// TIA Portal V16 export
// export: Created 2021-11-12T13:32:44.479513Z, ExportSetting WithDefaults, DisplayName Totally Integrated Automation Portal, DisplayVersion V16 Update 3, DisplayName TIA Portal Version Control Interface, DisplayVersion V16 Update 2, DisplayName TIA Portal Openness, DisplayVersion V16 Update 3, DisplayName SINAMICS Startdrive Advanced, DisplayVersion V16 Update 5, DisplayName SINAMICS Startdrive G130, G150, S120, S150, SINAMICS MV, S210, DisplayVersion V16 Update 5, DisplayName SINAMICS Startdrive G110M, G120, G120C, G120D, G120P, G115D, DisplayVersion V16 Update 5, DisplayName STEP 7 Professional, DisplayVersion V16 Update 3, DisplayName STEP 7 Safety, DisplayVersion V16, DisplayName WinCC UA Professional, DisplayVersion V16 Update 3
FUNCTION_BLOCK "StationBSN3"   // FB46, LAD
{ S7_Optimized_Access := 'TRUE' }
VERSION : 0.1
// stored: AutoNumber true, IsIECCheckEnabled false, IsRetainMemResEnabled false, MemoryReserve 100, SetENOAutomatically false, UDAEnableTagReadback false
   VAR_INPUT
      IS_Inputs : "UDT_COMM_BSN3_CRS";   // Inputs from owens PLC
   END_VAR
   VAR_OUTPUT
      OS_Outputs : "UDT_COMM_CRS_BSN3";   // Outputs to owens PLC
      OS_Status : "UDT_BSN3_Status_specific";
   END_VAR
   VAR
      SF_TON_Tact : TON_TIME;
      SF_TON_1 { S7_SetPoint := 'True'} : TON_TIME;
      SF_Alarm1 : "STD_DI_Mon";
      SF_Alarm2 : "STD_DI_Mon";
      SF_Alarm3 : "STD_DI_Mon";
      SF_Alarm4 : "STD_DI_Mon";
      SF_Alarm5 : "STD_DI_Mon";
      SF_Alarm6 : "STD_DI_Mon";
      SF_Alarm7 : "STD_DI_Mon";
      SF_Alarm8 : "STD_DI_Mon";
      SF_CL01_Alarm { S7_SetPoint := 'True'} : "STD_DI_Mon";
      SF_CL01_Warning { S7_SetPoint := 'True'} : "STD_DI_Mon";
      SF_BoxPartCounter { S7_SetPoint := 'True'} : "STD_PartCounter";
      SS_Edge { S7_SetPoint := 'True'} : Array[0..15] of Bool;   // Edge evalution
      SS_ParamTemp : Struct
         PartType : Int;   // Production type
         SPBurnerHigh : Int := 0;   // setpoint burner high [mm]
         SPTempSetpointZ1 : Int := 0;   // temperature setpoint in zone 1 [°C]
         SPTempSetpointZ2 : Int := 0;   // temperature setpoint in zone 2 [°C]
         SPTempSetpointZ3 : Int := 0;   // temperature setpoint in zone 3 [°C]
         SPTempSetpointZ4 : Int := 0;   // temperature setpoint in zone 4 [°C]
         SPTempSetpointZ5 : Int := 0;   // temperature setpoint in zone 5 [°C]
         SPTempSetpointZ6 : Int := 0;   // temperature setpoint in zone 5 [°C]
         SPTempSetpointZ7 : Int := 0;   // temperature setpoint in zone 5 [°C]
         ActPartTime : Int;   // actual setpoint of time in furnace according to belt speed [min]
      END_STRUCT;
      SB1BoxExchangeReq { S7_SetPoint := 'True'} : Bool;
      SB1ReqBlockBeltMtion : Bool;   // Button request to block belt motion
      SB1ReqBlockBeltMtion_Aux : Bool;
      SB1ParamChanged : Bool;   // Production paramaters changed trigger
      ST_RunConv { S7_SetPoint := 'True'} : TOF_TIME;
   END_VAR
   VAR_TEMP
      TS_ParamTemp : Struct
         PartType : Int;   // Production type
         SPBurnerHigh : Int;   // setpoint burner high [mm]
         SPTempSetpointZ1 : Int;   // temperature setpoint in zone 1 [°C]
         SPTempSetpointZ2 : Int;   // temperature setpoint in zone 2 [°C]
         SPTempSetpointZ3 : Int;   // temperature setpoint in zone 3 [°C]
         SPTempSetpointZ4 : Int;   // temperature setpoint in zone 4 [°C]
         SPTempSetpointZ5 : Int;   // temperature setpoint in zone 5 [°C]
         SPTempSetpointZ6 : Int;   // temperature setpoint in zone 5 [°C]
         SPTempSetpointZ7 : Int;   // temperature setpoint in zone 5 [°C]
         ActPartTime : Int;   // actual setpoint of time in furnace according to belt speed [min]
      END_STRUCT;
      TI_NoOfParts : Int;   // Number of parts before press
      TB1BoxFull : Bool;   // Box is full
      TB1PwrOk : Bool;
      TB1BeltMtionBlock : Bool;   // Belt motion blocking
      TB1ReqBlockBeltMtion : Bool;
      TB1ReqOnePart : Bool;   // Request to eject one part
      TB1ReqAllParts : Bool;   // Request to eject all parts in row
      TB1SetParam : Bool;   // Set loaded parameters memory
   END_VAR
   VAR_TEMP   // added for the SCL form of the ladder/FBD networks
      _w1 : Bool;
      _w2 : Bool;
   END_VAR
BEGIN

REGION Network 1: Copy In/Out variables to temporary variables
END_REGION

REGION Network 2: *************** Alarms ***************
END_REGION

REGION Network 3: Power OK
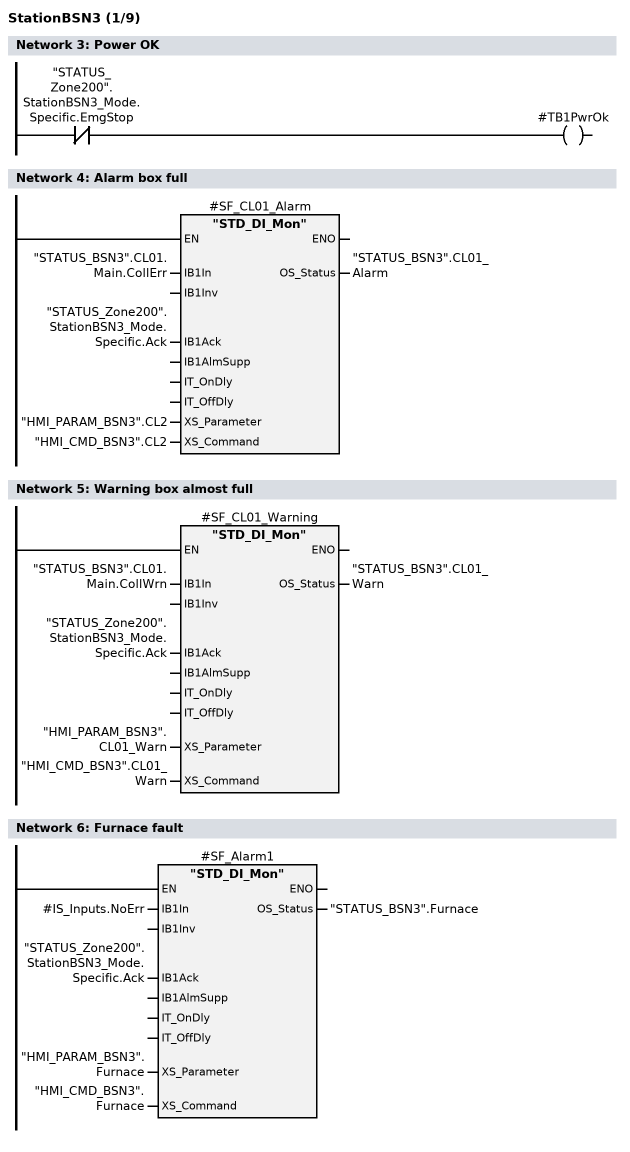
   RUNG wire#powerrail
      I_Contact( "STATUS_Zone200".StationBSN3_Mode.Specific.EmgStop )
      Coil( #TB1PwrOk )
   END_RUNG
   // the same network as SCL:
   #TB1PwrOk := NOT "STATUS_Zone200".StationBSN3_Mode.Specific.EmgStop;
END_REGION

REGION Network 4: Alarm box full
   RUNG wire#powerrail
      #SF_CL01_Alarm(IB1In := "STATUS_BSN3".CL01.Main.CollErr, IB1Inv :=, IB1Ack := "STATUS_Zone200".StationBSN3_Mode.Specific.Ack, IB1AlmSupp :=, IT_OnDly :=, IT_OffDly :=, XS_Parameter := "HMI_PARAM_BSN3".CL2, XS_Command := "HMI_CMD_BSN3".CL2, OS_Status => "STATUS_BSN3".CL01_Alarm)
   END_RUNG
   // the same network as SCL:
   #SF_CL01_Alarm(IB1In := "STATUS_BSN3".CL01.Main.CollErr,   // "STD_DI_Mon"
                  IB1Ack := "STATUS_Zone200".StationBSN3_Mode.Specific.Ack,
                  XS_Parameter := "HMI_PARAM_BSN3".CL2,
                  XS_Command := "HMI_CMD_BSN3".CL2,
                  OS_Status => "STATUS_BSN3".CL01_Alarm);
END_REGION

REGION Network 5: Warning box almost full
   RUNG wire#powerrail
      #SF_CL01_Warning(IB1In := "STATUS_BSN3".CL01.Main.CollWrn, IB1Inv :=, IB1Ack := "STATUS_Zone200".StationBSN3_Mode.Specific.Ack, IB1AlmSupp :=, IT_OnDly :=, IT_OffDly :=, XS_Parameter := "HMI_PARAM_BSN3".CL01_Warn, XS_Command := "HMI_CMD_BSN3".CL01_Warn, OS_Status => "STATUS_BSN3".CL01_Warn)
   END_RUNG
   // the same network as SCL:
   #SF_CL01_Warning(IB1In := "STATUS_BSN3".CL01.Main.CollWrn,   // "STD_DI_Mon"
                    IB1Ack := "STATUS_Zone200".StationBSN3_Mode.Specific.Ack,
                    XS_Parameter := "HMI_PARAM_BSN3".CL01_Warn,
                    XS_Command := "HMI_CMD_BSN3".CL01_Warn,
                    OS_Status => "STATUS_BSN3".CL01_Warn);
END_REGION

REGION Network 6: Furnace fault
   RUNG wire#powerrail
      #SF_Alarm1(IB1In := #IS_Inputs.NoErr, IB1Inv :=, IB1Ack := "STATUS_Zone200".StationBSN3_Mode.Specific.Ack, IB1AlmSupp :=, IT_OnDly :=, IT_OffDly :=, XS_Parameter := "HMI_PARAM_BSN3".Furnace, XS_Command := "HMI_CMD_BSN3".Furnace, OS_Status => "STATUS_BSN3".Furnace)
   END_RUNG
   // the same network as SCL:
   #SF_Alarm1(IB1In := #IS_Inputs.NoErr,   // "STD_DI_Mon"
              IB1Ack := "STATUS_Zone200".StationBSN3_Mode.Specific.Ack,
              XS_Parameter := "HMI_PARAM_BSN3".Furnace,
              XS_Command := "HMI_CMD_BSN3".Furnace,
              OS_Status => "STATUS_BSN3".Furnace);
END_REGION

REGION Network 7: Error in comunnication
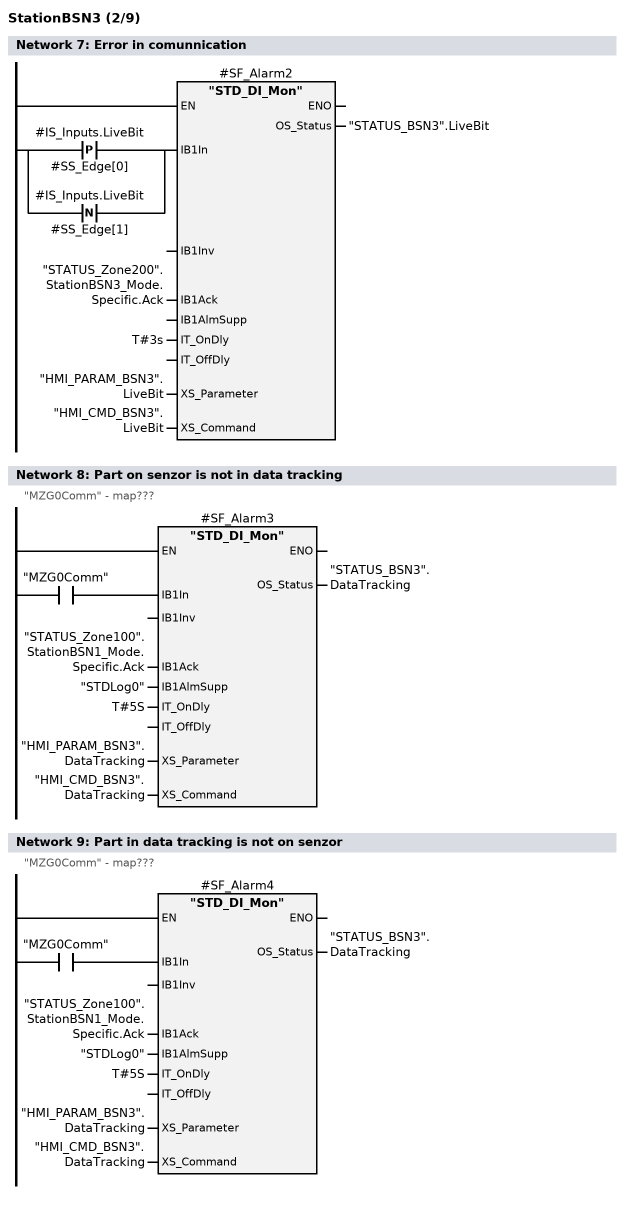
   RUNG wire#powerrail
      #SF_Alarm2(IB1In := wire#w1, IB1Inv :=, IB1Ack := "STATUS_Zone200".StationBSN3_Mode.Specific.Ack, IB1AlmSupp :=, IT_OnDly := T#3s, IT_OffDly :=, XS_Parameter := "HMI_PARAM_BSN3".LiveBit, XS_Command := "HMI_CMD_BSN3".LiveBit, OS_Status => "STATUS_BSN3".LiveBit)
   END_RUNG
   RUNG wire#powerrail
      P_Contact(operand := #IS_Inputs.LiveBit, bit := #SS_Edge[0])
   END_RUNG wire#w1
   RUNG wire#powerrail
      N_Contact(operand := #IS_Inputs.LiveBit, bit := #SS_Edge[1])
   END_RUNG wire#w1
   // the same network as SCL:
   #_w1 := #IS_Inputs.LiveBit AND NOT #SS_Edge[0];   // rising edge of #IS_Inputs.LiveBit
   #SS_Edge[0] := #IS_Inputs.LiveBit;
   #_w2 := NOT #IS_Inputs.LiveBit AND #SS_Edge[1];   // falling edge of #IS_Inputs.LiveBit
   #SS_Edge[1] := #IS_Inputs.LiveBit;
   #SF_Alarm2(IB1In := #_w1 OR #_w2,   // "STD_DI_Mon"
              IB1Ack := "STATUS_Zone200".StationBSN3_Mode.Specific.Ack,
              IT_OnDly := T#3s,
              XS_Parameter := "HMI_PARAM_BSN3".LiveBit,
              XS_Command := "HMI_CMD_BSN3".LiveBit,
              OS_Status => "STATUS_BSN3".LiveBit);
END_REGION

REGION Network 8: Part on senzor is not in data tracking
   // "MZG0Comm" - map???
   RUNG wire#powerrail
      #SF_Alarm3(IB1In := wire#w1, IB1Inv :=, IB1Ack := "STATUS_Zone100".StationBSN1_Mode.Specific.Ack, IB1AlmSupp := "STDLog0", IT_OnDly := T#5S, IT_OffDly :=, XS_Parameter := "HMI_PARAM_BSN3".DataTracking, XS_Command := "HMI_CMD_BSN3".DataTracking, OS_Status => "STATUS_BSN3".DataTracking)
   END_RUNG
   RUNG wire#powerrail
      Contact( "MZG0Comm" )
   END_RUNG wire#w1
   // the same network as SCL:
   #SF_Alarm3(IB1In := "MZG0Comm",   // "STD_DI_Mon"
              IB1Ack := "STATUS_Zone100".StationBSN1_Mode.Specific.Ack,
              IB1AlmSupp := "STDLog0",
              IT_OnDly := T#5S,
              XS_Parameter := "HMI_PARAM_BSN3".DataTracking,
              XS_Command := "HMI_CMD_BSN3".DataTracking,
              OS_Status => "STATUS_BSN3".DataTracking);
END_REGION

REGION Network 9: Part in data tracking is not on senzor
   // "MZG0Comm" - map???
   RUNG wire#powerrail
      #SF_Alarm4(IB1In := wire#w1, IB1Inv :=, IB1Ack := "STATUS_Zone100".StationBSN1_Mode.Specific.Ack, IB1AlmSupp := "STDLog0", IT_OnDly := T#5S, IT_OffDly :=, XS_Parameter := "HMI_PARAM_BSN3".DataTracking, XS_Command := "HMI_CMD_BSN3".DataTracking, OS_Status => "STATUS_BSN3".DataTracking)
   END_RUNG
   RUNG wire#powerrail
      Contact( "MZG0Comm" )
   END_RUNG wire#w1
   // the same network as SCL:
   #SF_Alarm4(IB1In := "MZG0Comm",   // "STD_DI_Mon"
              IB1Ack := "STATUS_Zone100".StationBSN1_Mode.Specific.Ack,
              IB1AlmSupp := "STDLog0",
              IT_OnDly := T#5S,
              XS_Parameter := "HMI_PARAM_BSN3".DataTracking,
              XS_Command := "HMI_CMD_BSN3".DataTracking,
              OS_Status => "STATUS_BSN3".DataTracking);
END_REGION

REGION Network 10: Alarm 9
   // timeout error from input to output
END_REGION

REGION Network 11: *************** States ***************
END_REGION

REGION Network 12: Temperature, belt extension, ejectors, belt movement
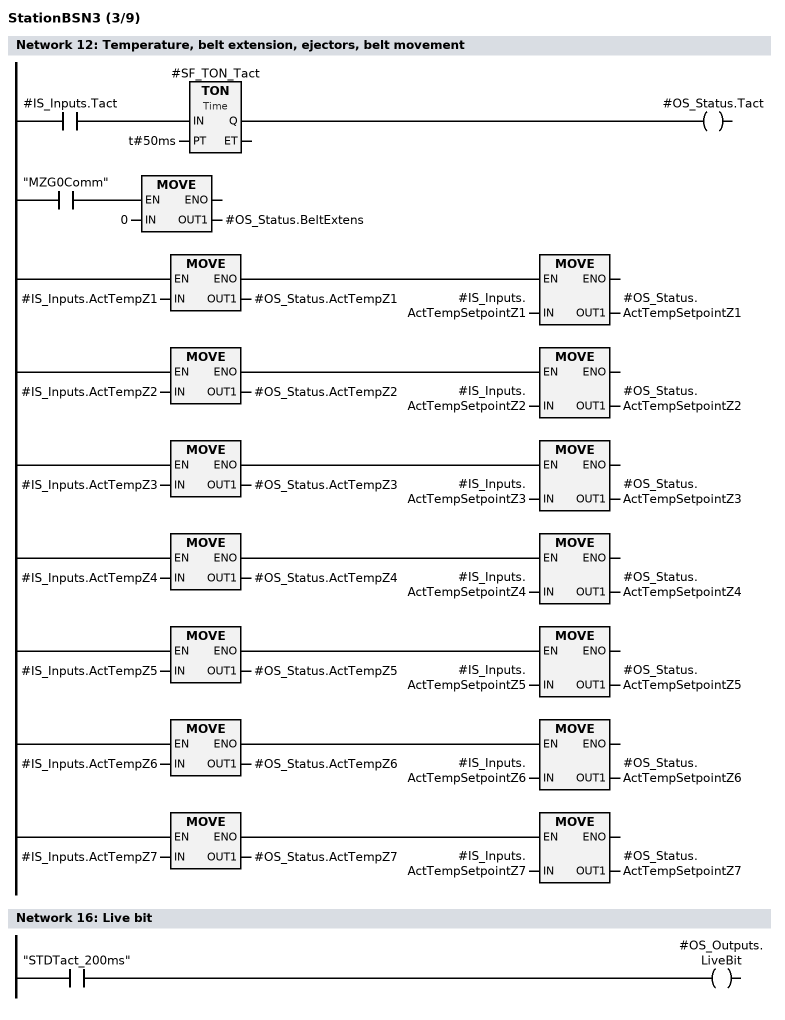
   RUNG wire#powerrail
      Contact( #IS_Inputs.Tact )
      { S7_Templates := "time_type := Time" } #SF_TON_Tact.TON(pt := t#50ms, et =>)
      Coil( #OS_Status.Tact )
   END_RUNG
   RUNG wire#powerrail
      Contact( "MZG0Comm" )
      Move(in := 0, out1 => #OS_Status.BeltExtens)
   END_RUNG
   RUNG wire#powerrail
      Move(in := #IS_Inputs.ActTempZ1, out1 => #OS_Status.ActTempZ1)
      Move(in := #IS_Inputs.ActTempSetpointZ1, out1 => #OS_Status.ActTempSetpointZ1)
   END_RUNG
   RUNG wire#powerrail
      Move(in := #IS_Inputs.ActTempZ2, out1 => #OS_Status.ActTempZ2)
      Move(in := #IS_Inputs.ActTempSetpointZ2, out1 => #OS_Status.ActTempSetpointZ2)
   END_RUNG
   RUNG wire#powerrail
      Move(in := #IS_Inputs.ActTempZ3, out1 => #OS_Status.ActTempZ3)
      Move(in := #IS_Inputs.ActTempSetpointZ3, out1 => #OS_Status.ActTempSetpointZ3)
   END_RUNG
   RUNG wire#powerrail
      Move(in := #IS_Inputs.ActTempZ4, out1 => #OS_Status.ActTempZ4)
      Move(in := #IS_Inputs.ActTempSetpointZ4, out1 => #OS_Status.ActTempSetpointZ4)
   END_RUNG
   RUNG wire#powerrail
      Move(in := #IS_Inputs.ActTempZ5, out1 => #OS_Status.ActTempZ5)
      Move(in := #IS_Inputs.ActTempSetpointZ5, out1 => #OS_Status.ActTempSetpointZ5)
   END_RUNG
   RUNG wire#powerrail
      Move(in := #IS_Inputs.ActTempZ6, out1 => #OS_Status.ActTempZ6)
      Move(in := #IS_Inputs.ActTempSetpointZ6, out1 => #OS_Status.ActTempSetpointZ6)
   END_RUNG
   RUNG wire#powerrail
      Move(in := #IS_Inputs.ActTempZ7, out1 => #OS_Status.ActTempZ7)
      Move(in := #IS_Inputs.ActTempSetpointZ7, out1 => #OS_Status.ActTempSetpointZ7)
   END_RUNG
   // the same network as SCL:
   #SF_TON_Tact(IN := #IS_Inputs.Tact, PT := t#50ms);   // TON
   #OS_Status.Tact := #SF_TON_Tact.Q;
   IF "MZG0Comm" THEN #OS_Status.BeltExtens := 0; END_IF;
   #OS_Status.ActTempZ1 := #IS_Inputs.ActTempZ1;
   #OS_Status.ActTempSetpointZ1 := #IS_Inputs.ActTempSetpointZ1;
   #OS_Status.ActTempZ2 := #IS_Inputs.ActTempZ2;
   #OS_Status.ActTempSetpointZ2 := #IS_Inputs.ActTempSetpointZ2;
   #OS_Status.ActTempZ3 := #IS_Inputs.ActTempZ3;
   #OS_Status.ActTempSetpointZ3 := #IS_Inputs.ActTempSetpointZ3;
   #OS_Status.ActTempZ4 := #IS_Inputs.ActTempZ4;
   #OS_Status.ActTempSetpointZ4 := #IS_Inputs.ActTempSetpointZ4;
   #OS_Status.ActTempZ5 := #IS_Inputs.ActTempZ5;
   #OS_Status.ActTempSetpointZ5 := #IS_Inputs.ActTempSetpointZ5;
   #OS_Status.ActTempZ6 := #IS_Inputs.ActTempZ6;
   #OS_Status.ActTempSetpointZ6 := #IS_Inputs.ActTempSetpointZ6;
   #OS_Status.ActTempZ7 := #IS_Inputs.ActTempZ7;
   #OS_Status.ActTempSetpointZ7 := #IS_Inputs.ActTempSetpointZ7;
END_REGION

REGION Network 13: Furnace part counter
END_REGION

REGION Network 14: Output conveyor part counter
END_REGION

REGION Network 15: ***************Interface to furnace ***************
END_REGION

REGION Network 16: Live bit
   RUNG wire#powerrail
      Contact( "STDTact_200ms" )
      Coil( #OS_Outputs.LiveBit )
   END_RUNG
   // the same network as SCL:
   #OS_Outputs.LiveBit := "STDTact_200ms";
END_REGION

REGION Network 17: Run conveyour
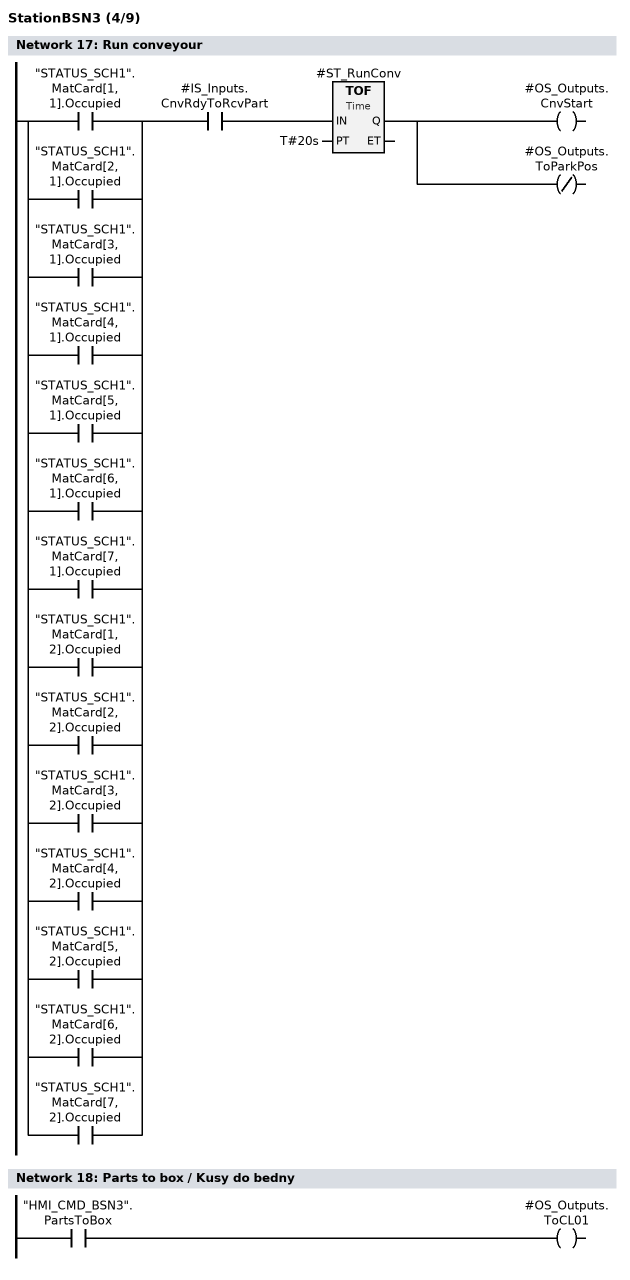
   RUNG wire#powerrail
      Contact( "STATUS_SCH1".MatCard[1, 1].Occupied )
      wire#w1
      Contact( #IS_Inputs.CnvRdyToRcvPart )
      { S7_Templates := "time_type := Time" } #ST_RunConv.TOF(pt := T#20s, et =>)
      wire#w2
      Coil( #OS_Outputs.CnvStart )
   END_RUNG
   RUNG wire#powerrail
      Contact( "STATUS_SCH1".MatCard[2, 1].Occupied )
   END_RUNG wire#w1
   RUNG wire#powerrail
      Contact( "STATUS_SCH1".MatCard[3, 1].Occupied )
   END_RUNG wire#w1
   RUNG wire#powerrail
      Contact( "STATUS_SCH1".MatCard[4, 1].Occupied )
   END_RUNG wire#w1
   RUNG wire#powerrail
      Contact( "STATUS_SCH1".MatCard[5, 1].Occupied )
   END_RUNG wire#w1
   RUNG wire#powerrail
      Contact( "STATUS_SCH1".MatCard[6, 1].Occupied )
   END_RUNG wire#w1
   RUNG wire#powerrail
      Contact( "STATUS_SCH1".MatCard[7, 1].Occupied )
   END_RUNG wire#w1
   RUNG wire#powerrail
      Contact( "STATUS_SCH1".MatCard[1, 2].Occupied )
   END_RUNG wire#w1
   RUNG wire#powerrail
      Contact( "STATUS_SCH1".MatCard[2, 2].Occupied )
   END_RUNG wire#w1
   RUNG wire#powerrail
      Contact( "STATUS_SCH1".MatCard[3, 2].Occupied )
   END_RUNG wire#w1
   RUNG wire#powerrail
      Contact( "STATUS_SCH1".MatCard[4, 2].Occupied )
   END_RUNG wire#w1
   RUNG wire#powerrail
      Contact( "STATUS_SCH1".MatCard[5, 2].Occupied )
   END_RUNG wire#w1
   RUNG wire#powerrail
      Contact( "STATUS_SCH1".MatCard[6, 2].Occupied )
   END_RUNG wire#w1
   RUNG wire#powerrail
      Contact( "STATUS_SCH1".MatCard[7, 2].Occupied )
   END_RUNG wire#w1
   RUNG wire#w2
      I_Coil( #OS_Outputs.ToParkPos )
   END_RUNG
   // the same network as SCL:
   #ST_RunConv(IN := ("STATUS_SCH1".MatCard[1, 1].Occupied OR "STATUS_SCH1".MatCard[2, 1].Occupied OR "STATUS_SCH1".MatCard[3, 1].Occupied OR "STATUS_SCH1".MatCard[4, 1].Occupied OR "STATUS_SCH1".MatCard[5, 1].Occupied OR "STATUS_SCH1".MatCard[6, 1].Occupied OR "STATUS_SCH1".MatCard[7, 1].Occupied OR "STATUS_SCH1".MatCard[1, 2].Occupied OR "STATUS_SCH1".MatCard[2, 2].Occupied OR "STATUS_SCH1".MatCard[3, 2].Occupied OR "STATUS_SCH1".MatCard[4, 2].Occupied OR "STATUS_SCH1".MatCard[5, 2].Occupied OR "STATUS_SCH1".MatCard[6, 2].Occupied OR "STATUS_SCH1".MatCard[7, 2].Occupied) AND #IS_Inputs.CnvRdyToRcvPart,   // TOF
               PT := T#20s);
   #OS_Outputs.CnvStart := #ST_RunConv.Q;
   #OS_Outputs.ToParkPos := NOT #ST_RunConv.Q;
END_REGION

REGION Network 18: Parts to box / Kusy do bedny
   RUNG wire#powerrail
      Contact( "HMI_CMD_BSN3".PartsToBox )
      Coil( #OS_Outputs.ToCL01 )
   END_RUNG
   // the same network as SCL:
   #OS_Outputs.ToCL01 := "HMI_CMD_BSN3".PartsToBox;
END_REGION

REGION Network 19: ************** Production parameters***************
END_REGION

REGION Network 20: Production parameters conversion
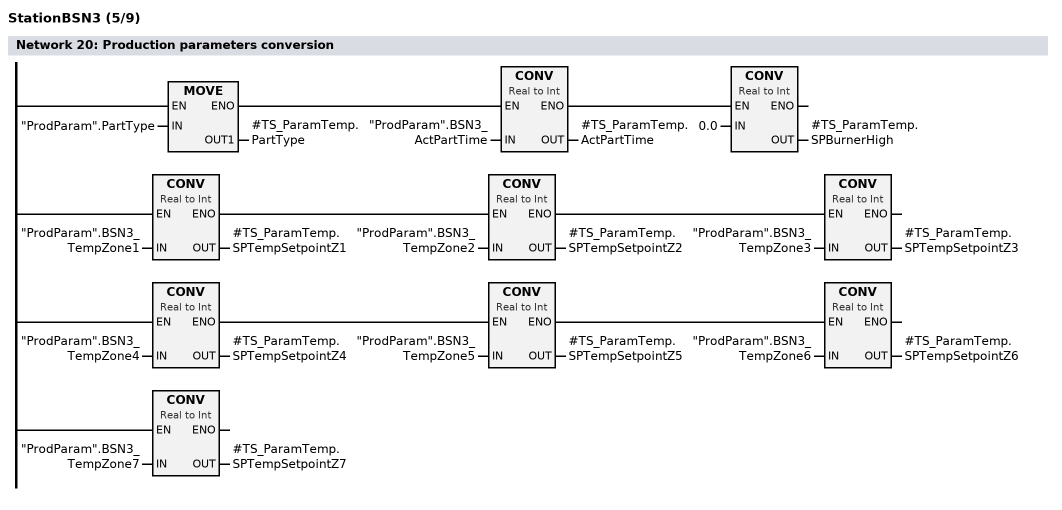
   RUNG wire#powerrail
      Move(in := "ProdParam".PartType, out1 => #TS_ParamTemp.PartType)
      { S7_Templates := "[SrcType := Real, DestType := Int]" } Convert(in := "ProdParam".BSN3_ActPartTime, out => #TS_ParamTemp.ActPartTime)
      { S7_Templates := "[SrcType := Real, DestType := Int]" } Convert(in := 0.0, out => #TS_ParamTemp.SPBurnerHigh)
   END_RUNG
   RUNG wire#powerrail
      { S7_Templates := "[SrcType := Real, DestType := Int]" } Convert(in := "ProdParam".BSN3_TempZone1, out => #TS_ParamTemp.SPTempSetpointZ1)
      { S7_Templates := "[SrcType := Real, DestType := Int]" } Convert(in := "ProdParam".BSN3_TempZone2, out => #TS_ParamTemp.SPTempSetpointZ2)
      { S7_Templates := "[SrcType := Real, DestType := Int]" } Convert(in := "ProdParam".BSN3_TempZone3, out => #TS_ParamTemp.SPTempSetpointZ3)
   END_RUNG
   RUNG wire#powerrail
      { S7_Templates := "[SrcType := Real, DestType := Int]" } Convert(in := "ProdParam".BSN3_TempZone4, out => #TS_ParamTemp.SPTempSetpointZ4)
      { S7_Templates := "[SrcType := Real, DestType := Int]" } Convert(in := "ProdParam".BSN3_TempZone5, out => #TS_ParamTemp.SPTempSetpointZ5)
      { S7_Templates := "[SrcType := Real, DestType := Int]" } Convert(in := "ProdParam".BSN3_TempZone6, out => #TS_ParamTemp.SPTempSetpointZ6)
   END_RUNG
   RUNG wire#powerrail
      { S7_Templates := "[SrcType := Real, DestType := Int]" } Convert(in := "ProdParam".BSN3_TempZone7, out => #TS_ParamTemp.SPTempSetpointZ7)
   END_RUNG
   // the same network as SCL:
   #TS_ParamTemp.PartType := "ProdParam".PartType;
   #TS_ParamTemp.ActPartTime := REAL_TO_INT("ProdParam".BSN3_ActPartTime);
   #TS_ParamTemp.SPBurnerHigh := REAL_TO_INT(0.0);
   #TS_ParamTemp.SPTempSetpointZ1 := REAL_TO_INT("ProdParam".BSN3_TempZone1);
   #TS_ParamTemp.SPTempSetpointZ2 := REAL_TO_INT("ProdParam".BSN3_TempZone2);
   #TS_ParamTemp.SPTempSetpointZ3 := REAL_TO_INT("ProdParam".BSN3_TempZone3);
   #TS_ParamTemp.SPTempSetpointZ4 := REAL_TO_INT("ProdParam".BSN3_TempZone4);
   #TS_ParamTemp.SPTempSetpointZ5 := REAL_TO_INT("ProdParam".BSN3_TempZone5);
   #TS_ParamTemp.SPTempSetpointZ6 := REAL_TO_INT("ProdParam".BSN3_TempZone6);
   #TS_ParamTemp.SPTempSetpointZ7 := REAL_TO_INT("ProdParam".BSN3_TempZone7);
END_REGION

REGION Network 21: Production parameter changed trigger
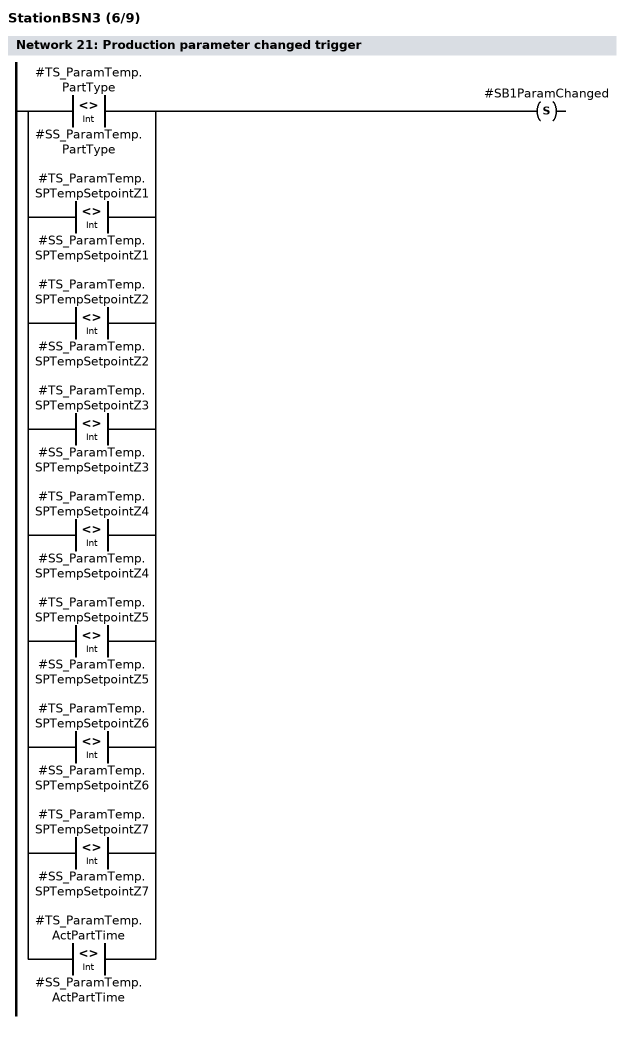
   RUNG wire#powerrail
      { S7_Templates := "SrcType := Int" } NE_Contact(in1 := #TS_ParamTemp.PartType, in2 := #SS_ParamTemp.PartType)
      wire#w1
      S_Coil( #SB1ParamChanged )
   END_RUNG
   RUNG wire#powerrail
      { S7_Templates := "SrcType := Int" } NE_Contact(in1 := #TS_ParamTemp.SPTempSetpointZ1, in2 := #SS_ParamTemp.SPTempSetpointZ1)
   END_RUNG wire#w1
   RUNG wire#powerrail
      { S7_Templates := "SrcType := Int" } NE_Contact(in1 := #TS_ParamTemp.SPTempSetpointZ2, in2 := #SS_ParamTemp.SPTempSetpointZ2)
   END_RUNG wire#w1
   RUNG wire#powerrail
      { S7_Templates := "SrcType := Int" } NE_Contact(in1 := #TS_ParamTemp.SPTempSetpointZ3, in2 := #SS_ParamTemp.SPTempSetpointZ3)
   END_RUNG wire#w1
   RUNG wire#powerrail
      { S7_Templates := "SrcType := Int" } NE_Contact(in1 := #TS_ParamTemp.SPTempSetpointZ4, in2 := #SS_ParamTemp.SPTempSetpointZ4)
   END_RUNG wire#w1
   RUNG wire#powerrail
      { S7_Templates := "SrcType := Int" } NE_Contact(in1 := #TS_ParamTemp.SPTempSetpointZ5, in2 := #SS_ParamTemp.SPTempSetpointZ5)
   END_RUNG wire#w1
   RUNG wire#powerrail
      { S7_Templates := "SrcType := Int" } NE_Contact(in1 := #TS_ParamTemp.SPTempSetpointZ6, in2 := #SS_ParamTemp.SPTempSetpointZ6)
   END_RUNG wire#w1
   RUNG wire#powerrail
      { S7_Templates := "SrcType := Int" } NE_Contact(in1 := #TS_ParamTemp.SPTempSetpointZ7, in2 := #SS_ParamTemp.SPTempSetpointZ7)
   END_RUNG wire#w1
   RUNG wire#powerrail
      { S7_Templates := "SrcType := Int" } NE_Contact(in1 := #TS_ParamTemp.ActPartTime, in2 := #SS_ParamTemp.ActPartTime)
   END_RUNG wire#w1
   // the same network as SCL:
   IF (#TS_ParamTemp.PartType <> #SS_ParamTemp.PartType) OR (#TS_ParamTemp.SPTempSetpointZ1 <> #SS_ParamTemp.SPTempSetpointZ1) OR (#TS_ParamTemp.SPTempSetpointZ2 <> #SS_ParamTemp.SPTempSetpointZ2) OR (#TS_ParamTemp.SPTempSetpointZ3 <> #SS_ParamTemp.SPTempSetpointZ3) OR (#TS_ParamTemp.SPTempSetpointZ4 <> #SS_ParamTemp.SPTempSetpointZ4) OR (#TS_ParamTemp.SPTempSetpointZ5 <> #SS_ParamTemp.SPTempSetpointZ5) OR (#TS_ParamTemp.SPTempSetpointZ6 <> #SS_ParamTemp.SPTempSetpointZ6) OR (#TS_ParamTemp.SPTempSetpointZ7 <> #SS_ParamTemp.SPTempSetpointZ7) OR (#TS_ParamTemp.ActPartTime <> #SS_ParamTemp.ActPartTime) THEN
       #SB1ParamChanged := TRUE;
   END_IF;
END_REGION

REGION Network 22: Production parameters values memory for next cycle evaluation
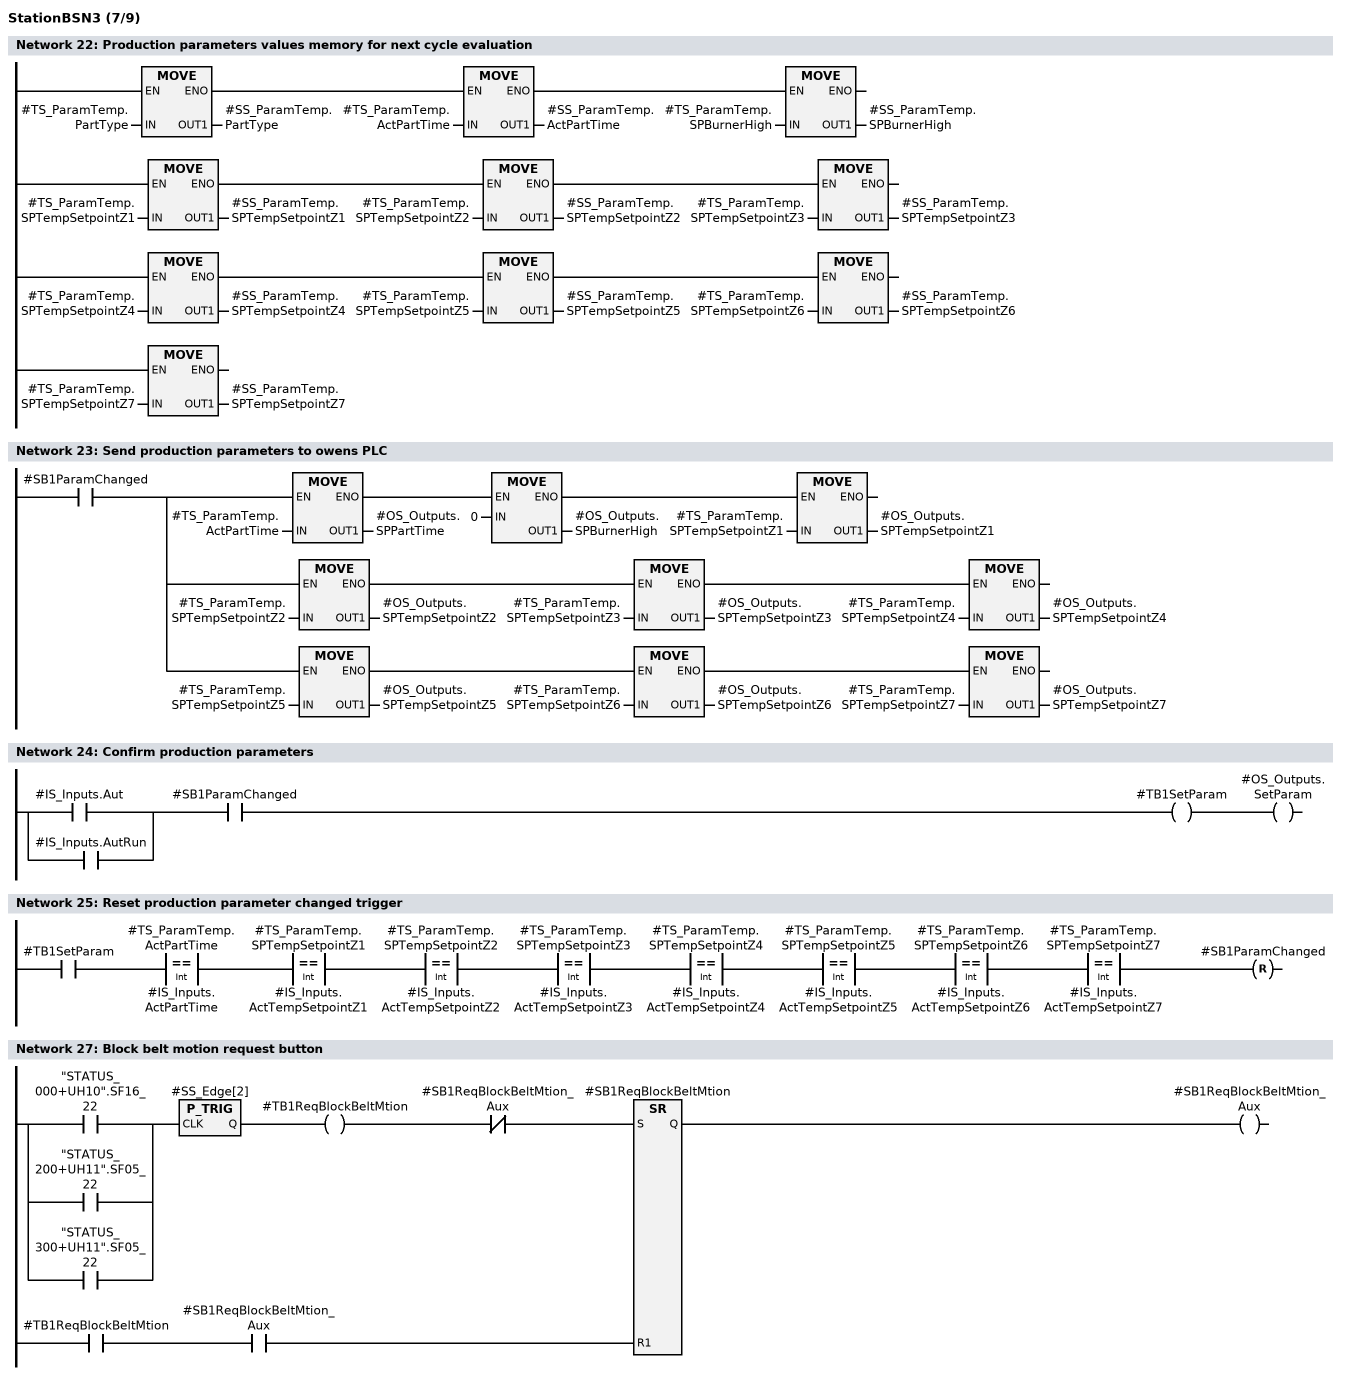
   RUNG wire#powerrail
      Move(in := #TS_ParamTemp.PartType, out1 => #SS_ParamTemp.PartType)
      Move(in := #TS_ParamTemp.ActPartTime, out1 => #SS_ParamTemp.ActPartTime)
      Move(in := #TS_ParamTemp.SPBurnerHigh, out1 => #SS_ParamTemp.SPBurnerHigh)
   END_RUNG
   RUNG wire#powerrail
      Move(in := #TS_ParamTemp.SPTempSetpointZ1, out1 => #SS_ParamTemp.SPTempSetpointZ1)
      Move(in := #TS_ParamTemp.SPTempSetpointZ2, out1 => #SS_ParamTemp.SPTempSetpointZ2)
      Move(in := #TS_ParamTemp.SPTempSetpointZ3, out1 => #SS_ParamTemp.SPTempSetpointZ3)
   END_RUNG
   RUNG wire#powerrail
      Move(in := #TS_ParamTemp.SPTempSetpointZ4, out1 => #SS_ParamTemp.SPTempSetpointZ4)
      Move(in := #TS_ParamTemp.SPTempSetpointZ5, out1 => #SS_ParamTemp.SPTempSetpointZ5)
      Move(in := #TS_ParamTemp.SPTempSetpointZ6, out1 => #SS_ParamTemp.SPTempSetpointZ6)
   END_RUNG
   RUNG wire#powerrail
      Move(in := #TS_ParamTemp.SPTempSetpointZ7, out1 => #SS_ParamTemp.SPTempSetpointZ7)
   END_RUNG
   // the same network as SCL:
   #SS_ParamTemp.PartType := #TS_ParamTemp.PartType;
   #SS_ParamTemp.ActPartTime := #TS_ParamTemp.ActPartTime;
   #SS_ParamTemp.SPBurnerHigh := #TS_ParamTemp.SPBurnerHigh;
   #SS_ParamTemp.SPTempSetpointZ1 := #TS_ParamTemp.SPTempSetpointZ1;
   #SS_ParamTemp.SPTempSetpointZ2 := #TS_ParamTemp.SPTempSetpointZ2;
   #SS_ParamTemp.SPTempSetpointZ3 := #TS_ParamTemp.SPTempSetpointZ3;
   #SS_ParamTemp.SPTempSetpointZ4 := #TS_ParamTemp.SPTempSetpointZ4;
   #SS_ParamTemp.SPTempSetpointZ5 := #TS_ParamTemp.SPTempSetpointZ5;
   #SS_ParamTemp.SPTempSetpointZ6 := #TS_ParamTemp.SPTempSetpointZ6;
   #SS_ParamTemp.SPTempSetpointZ7 := #TS_ParamTemp.SPTempSetpointZ7;
END_REGION

REGION Network 23: Send production parameters to owens PLC
   RUNG wire#powerrail
      Contact( #SB1ParamChanged )
      wire#w1
      Move(in := #TS_ParamTemp.ActPartTime, out1 => #OS_Outputs.SPPartTime)
      Move(in := 0, out1 => #OS_Outputs.SPBurnerHigh)
      Move(in := #TS_ParamTemp.SPTempSetpointZ1, out1 => #OS_Outputs.SPTempSetpointZ1)
   END_RUNG
   RUNG wire#w1
      Move(in := #TS_ParamTemp.SPTempSetpointZ2, out1 => #OS_Outputs.SPTempSetpointZ2)
      Move(in := #TS_ParamTemp.SPTempSetpointZ3, out1 => #OS_Outputs.SPTempSetpointZ3)
      Move(in := #TS_ParamTemp.SPTempSetpointZ4, out1 => #OS_Outputs.SPTempSetpointZ4)
   END_RUNG
   RUNG wire#w1
      Move(in := #TS_ParamTemp.SPTempSetpointZ5, out1 => #OS_Outputs.SPTempSetpointZ5)
      Move(in := #TS_ParamTemp.SPTempSetpointZ6, out1 => #OS_Outputs.SPTempSetpointZ6)
      Move(in := #TS_ParamTemp.SPTempSetpointZ7, out1 => #OS_Outputs.SPTempSetpointZ7)
   END_RUNG
   // the same network as SCL:
   IF #SB1ParamChanged THEN
       #OS_Outputs.SPPartTime := #TS_ParamTemp.ActPartTime;
       #OS_Outputs.SPBurnerHigh := 0;
       #OS_Outputs.SPTempSetpointZ1 := #TS_ParamTemp.SPTempSetpointZ1;
       #OS_Outputs.SPTempSetpointZ2 := #TS_ParamTemp.SPTempSetpointZ2;
       #OS_Outputs.SPTempSetpointZ3 := #TS_ParamTemp.SPTempSetpointZ3;
       #OS_Outputs.SPTempSetpointZ4 := #TS_ParamTemp.SPTempSetpointZ4;
       #OS_Outputs.SPTempSetpointZ5 := #TS_ParamTemp.SPTempSetpointZ5;
       #OS_Outputs.SPTempSetpointZ6 := #TS_ParamTemp.SPTempSetpointZ6;
       #OS_Outputs.SPTempSetpointZ7 := #TS_ParamTemp.SPTempSetpointZ7;
   END_IF;
END_REGION

REGION Network 24: Confirm production parameters
   RUNG wire#powerrail
      Contact( #IS_Inputs.Aut )
      wire#w1
      Contact( #SB1ParamChanged )
      Coil( #TB1SetParam )
      Coil( #OS_Outputs.SetParam )
   END_RUNG
   RUNG wire#powerrail
      Contact( #IS_Inputs.AutRun )
   END_RUNG wire#w1
   // the same network as SCL:
   #TB1SetParam := (#IS_Inputs.Aut OR #IS_Inputs.AutRun) AND #SB1ParamChanged;
   #OS_Outputs.SetParam := #TB1SetParam;
END_REGION

REGION Network 25: Reset production parameter changed trigger
   RUNG wire#powerrail
      Contact( #TB1SetParam )
      { S7_Templates := "SrcType := Int" } EQ_Contact(in1 := #TS_ParamTemp.ActPartTime, in2 := #IS_Inputs.ActPartTime)
      { S7_Templates := "SrcType := Int" } EQ_Contact(in1 := #TS_ParamTemp.SPTempSetpointZ1, in2 := #IS_Inputs.ActTempSetpointZ1)
      { S7_Templates := "SrcType := Int" } EQ_Contact(in1 := #TS_ParamTemp.SPTempSetpointZ2, in2 := #IS_Inputs.ActTempSetpointZ2)
      { S7_Templates := "SrcType := Int" } EQ_Contact(in1 := #TS_ParamTemp.SPTempSetpointZ3, in2 := #IS_Inputs.ActTempSetpointZ3)
      { S7_Templates := "SrcType := Int" } EQ_Contact(in1 := #TS_ParamTemp.SPTempSetpointZ4, in2 := #IS_Inputs.ActTempSetpointZ4)
      { S7_Templates := "SrcType := Int" } EQ_Contact(in1 := #TS_ParamTemp.SPTempSetpointZ5, in2 := #IS_Inputs.ActTempSetpointZ5)
      { S7_Templates := "SrcType := Int" } EQ_Contact(in1 := #TS_ParamTemp.SPTempSetpointZ6, in2 := #IS_Inputs.ActTempSetpointZ6)
      { S7_Templates := "SrcType := Int" } EQ_Contact(in1 := #TS_ParamTemp.SPTempSetpointZ7, in2 := #IS_Inputs.ActTempSetpointZ7)
      R_Coil( #SB1ParamChanged )
   END_RUNG
   // the same network as SCL:
   IF #TB1SetParam AND (#TS_ParamTemp.ActPartTime = #IS_Inputs.ActPartTime) AND (#TS_ParamTemp.SPTempSetpointZ1 = #IS_Inputs.ActTempSetpointZ1) AND (#TS_ParamTemp.SPTempSetpointZ2 = #IS_Inputs.ActTempSetpointZ2) AND (#TS_ParamTemp.SPTempSetpointZ3 = #IS_Inputs.ActTempSetpointZ3) AND (#TS_ParamTemp.SPTempSetpointZ4 = #IS_Inputs.ActTempSetpointZ4) AND (#TS_ParamTemp.SPTempSetpointZ5 = #IS_Inputs.ActTempSetpointZ5) AND (#TS_ParamTemp.SPTempSetpointZ6 = #IS_Inputs.ActTempSetpointZ6) AND (#TS_ParamTemp.SPTempSetpointZ7 = #IS_Inputs.ActTempSetpointZ7) THEN
       #SB1ParamChanged := FALSE;
   END_IF;
END_REGION

REGION Network 26: ***************Belt ***************
END_REGION

REGION Network 27: Block belt motion request button
   RUNG wire#powerrail
      Contact( "STATUS_000+UH10".SF16_22 )
      wire#w1
      P_Trig( #SS_Edge[2] )
      Coil( #TB1ReqBlockBeltMtion )
      I_Contact( #SB1ReqBlockBeltMtion_Aux )
      S_SR(operand := #SB1ReqBlockBeltMtion, r1 := wire#w2)
      Coil( #SB1ReqBlockBeltMtion_Aux )
   END_RUNG
   RUNG wire#powerrail
      Contact( "STATUS_200+UH11".SF05_22 )
   END_RUNG wire#w1
   RUNG wire#powerrail
      Contact( "STATUS_300+UH11".SF05_22 )
   END_RUNG wire#w1
   RUNG wire#powerrail
      Contact( #TB1ReqBlockBeltMtion )
      Contact( #SB1ReqBlockBeltMtion_Aux )
   END_RUNG wire#w2
   // the same network as SCL:
   #_w1 := "STATUS_000+UH10".SF16_22 OR "STATUS_200+UH11".SF05_22 OR "STATUS_300+UH11".SF05_22;
   #_w2 := #_w1 AND NOT #SS_Edge[2];   // rising edge
   #SS_Edge[2] := #_w1;
   #TB1ReqBlockBeltMtion := #_w2;
   IF #_w2 AND NOT #SB1ReqBlockBeltMtion_Aux THEN
       #SB1ReqBlockBeltMtion := TRUE;   // SR flip-flop
   END_IF;
   IF #TB1ReqBlockBeltMtion AND #SB1ReqBlockBeltMtion_Aux THEN #SB1ReqBlockBeltMtion := FALSE; END_IF;
   #SB1ReqBlockBeltMtion_Aux := #SB1ReqBlockBeltMtion;
END_REGION

REGION Network 28: Blocking belt motion - summary
   // "JSA0Comm" - parts in owen
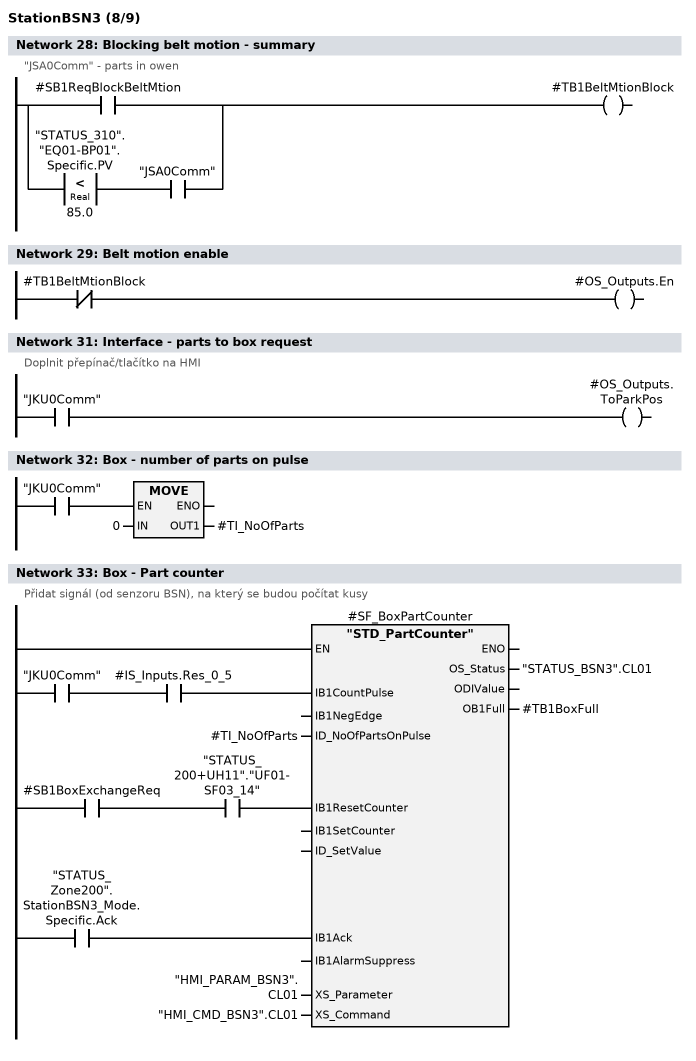
   RUNG wire#powerrail
      Contact( #SB1ReqBlockBeltMtion )
      wire#w1
      Coil( #TB1BeltMtionBlock )
   END_RUNG
   RUNG wire#powerrail
      { S7_Templates := "SrcType := Real" } LT_Contact(in1 := "STATUS_310"."EQ01-BP01".Specific.PV, in2 := 85.0)
      Contact( "JSA0Comm" )
   END_RUNG wire#w1
   // the same network as SCL:
   #TB1BeltMtionBlock := #SB1ReqBlockBeltMtion OR (("STATUS_310"."EQ01-BP01".Specific.PV < 85.0) AND "JSA0Comm");
END_REGION

REGION Network 29: Belt motion enable
   RUNG wire#powerrail
      I_Contact( #TB1BeltMtionBlock )
      Coil( #OS_Outputs.En )
   END_RUNG
   // the same network as SCL:
   #OS_Outputs.En := NOT #TB1BeltMtionBlock;
END_REGION

REGION Network 30: *************** Box ***************
END_REGION

REGION Network 31: Interface - parts to box request
   // Doplnit přepínač/tlačítko na HMI
   RUNG wire#powerrail
      Contact( "JKU0Comm" )
      Coil( #OS_Outputs.ToParkPos )
   END_RUNG
   // the same network as SCL:
   #OS_Outputs.ToParkPos := "JKU0Comm";
END_REGION

REGION Network 32: Box - number of parts on pulse
   RUNG wire#powerrail
      Contact( "JKU0Comm" )
      Move(in := 0, out1 => #TI_NoOfParts)
   END_RUNG
   // the same network as SCL:
   IF "JKU0Comm" THEN #TI_NoOfParts := 0; END_IF;
END_REGION

REGION Network 33: Box - Part counter
   // Přidat signál (od senzoru BSN), na který se budou počítat kusy
   RUNG wire#powerrail
      #SF_BoxPartCounter(IB1CountPulse := wire#w1, IB1ResetCounter := wire#w2, IB1Ack := wire#w3, IB1NegEdge :=, ID_NoOfPartsOnPulse := #TI_NoOfParts, IB1SetCounter :=, ID_SetValue :=, IB1AlarmSuppress :=, XS_Parameter := "HMI_PARAM_BSN3".CL01, XS_Command := "HMI_CMD_BSN3".CL01, OS_Status => "STATUS_BSN3".CL01, ODIValue =>, OB1Full => #TB1BoxFull)
   END_RUNG
   RUNG wire#powerrail
      Contact( "JKU0Comm" )
      Contact( #IS_Inputs.Res_0_5 )
   END_RUNG wire#w1
   RUNG wire#powerrail
      Contact( #SB1BoxExchangeReq )
      Contact( "STATUS_200+UH11"."UF01-SF03_14" )
   END_RUNG wire#w2
   RUNG wire#powerrail
      Contact( "STATUS_Zone200".StationBSN3_Mode.Specific.Ack )
   END_RUNG wire#w3
   // the same network as SCL:
   #SF_BoxPartCounter(IB1CountPulse := "JKU0Comm" AND #IS_Inputs.Res_0_5,   // "STD_PartCounter"
                      ID_NoOfPartsOnPulse := #TI_NoOfParts,
                      IB1ResetCounter := #SB1BoxExchangeReq AND "STATUS_200+UH11"."UF01-SF03_14",
                      IB1Ack := "STATUS_Zone200".StationBSN3_Mode.Specific.Ack,
                      XS_Parameter := "HMI_PARAM_BSN3".CL01,
                      XS_Command := "HMI_CMD_BSN3".CL01,
                      OS_Status => "STATUS_BSN3".CL01,
                      OB1Full => #TB1BoxFull);
END_REGION

REGION Network 34: Box - exchange request
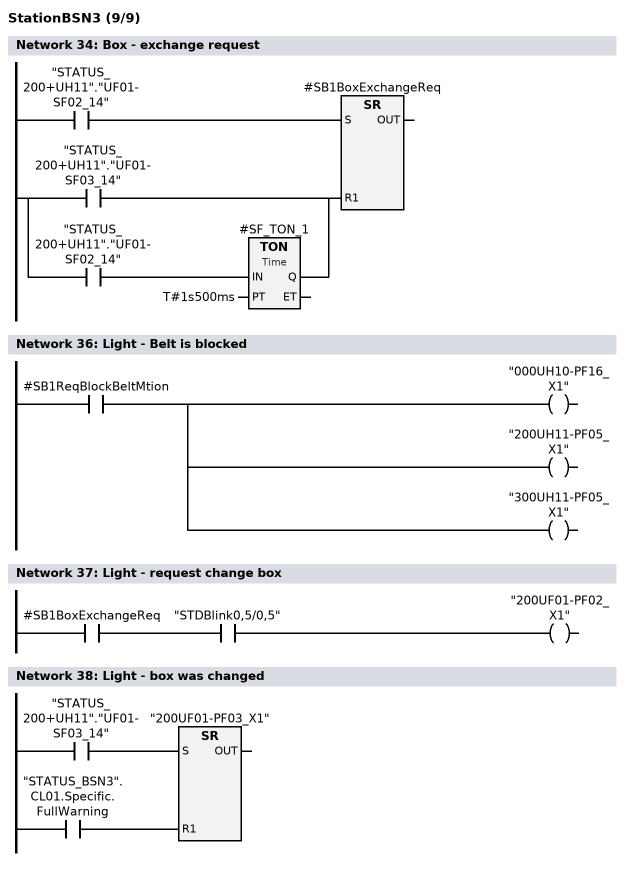
   RUNG wire#powerrail
      Contact( "STATUS_200+UH11"."UF01-SF02_14" )
      S_SR(operand := #SB1BoxExchangeReq, r1 := wire#w1)
   END_RUNG
   RUNG wire#powerrail
      Contact( "STATUS_200+UH11"."UF01-SF03_14" )
   END_RUNG wire#w1
   RUNG wire#powerrail
      Contact( "STATUS_200+UH11"."UF01-SF02_14" )
      { S7_Templates := "time_type := Time" } #SF_TON_1.TON(pt := T#1s500ms, et =>)
   END_RUNG wire#w1
   // the same network as SCL:
   #SF_TON_1(IN := "STATUS_200+UH11"."UF01-SF02_14", PT := T#1s500ms);   // TON
   IF "STATUS_200+UH11"."UF01-SF02_14" THEN
       #SB1BoxExchangeReq := TRUE;   // SR flip-flop
   END_IF;
   IF "STATUS_200+UH11"."UF01-SF03_14" OR #SF_TON_1.Q THEN #SB1BoxExchangeReq := FALSE; END_IF;
END_REGION

REGION Network 35: ************** Signalization ***************
END_REGION

REGION Network 36: Light - Belt is blocked
   RUNG wire#powerrail
      Contact( #SB1ReqBlockBeltMtion )
      wire#w1
      Coil( "000UH10-PF16_X1" )
   END_RUNG
   RUNG wire#w1
      Coil( "200UH11-PF05_X1" )
   END_RUNG
   RUNG wire#w1
      Coil( "300UH11-PF05_X1" )
   END_RUNG
   // the same network as SCL:
   "000UH10-PF16_X1" := #SB1ReqBlockBeltMtion;
   "200UH11-PF05_X1" := #SB1ReqBlockBeltMtion;
   "300UH11-PF05_X1" := #SB1ReqBlockBeltMtion;
END_REGION

REGION Network 37: Light - request change box
   RUNG wire#powerrail
      Contact( #SB1BoxExchangeReq )
      Contact( "STDBlink0,5/0,5" )
      Coil( "200UF01-PF02_X1" )
   END_RUNG
   // the same network as SCL:
   "200UF01-PF02_X1" := #SB1BoxExchangeReq AND "STDBlink0,5/0,5";
END_REGION

REGION Network 38: Light - box was changed
   RUNG wire#powerrail
      Contact( "STATUS_200+UH11"."UF01-SF03_14" )
      S_SR(operand := "200UF01-PF03_X1", r1 := wire#w1)
   END_RUNG
   RUNG wire#powerrail
      Contact( "STATUS_BSN3".CL01.Specific.FullWarning )
   END_RUNG wire#w1
   // the same network as SCL:
   IF "STATUS_200+UH11"."UF01-SF03_14" THEN
       "200UF01-PF03_X1" := TRUE;   // SR flip-flop
   END_IF;
   IF "STATUS_BSN3".CL01.Specific.FullWarning THEN "200UF01-PF03_X1" := FALSE; END_IF;
END_REGION

REGION Network 39: ************** Outputs ***************
END_REGION

REGION Network 40: Copy temporary variables to in/out variables
END_REGION
END_FUNCTION_BLOCK
